{attribute 'qualified_only'}
//{attribute 'strict'}
TYPE E_SM_ERROR :
(
	OK					:= 0,
	HW_NOT_OP,			
	WRONG_CMD,			
	INIT_FAILURE,		

	NOT_INITIALISED		:= 90,
	ZERO_POINTER		:= 100	// Simulator error
);
END_TYPE

(* stored: Version 1.1.0.1, ProductVersion 3.1.4022.16
   DUT E_SM_ERROR: Id {6375cba0-0d70-41e3-b006-e02157de4634} *)
